{attribute 'GeneratedUsingTerminal: KL2819'}
{attribute addProperty BoxType "KL2819"}
{attribute addProperty Id "Channel_1AT %Q*Channel_2EC3E8CA0"}
{attribute addProperty CRC "685127745"}
{attribute addProperty Size "0"}
TYPE KL2819_28D63841 :
STRUCT
	{attribute addProperty Name "Channel_1"}
	Channel_1 : Channel_2EC3E8CA;
END_STRUCT
END_TYPE

(* stored: Version 1.2.0.0, ProductVersion 3.1.4024.9
   DUT KL2819_28D63841: Id {c018a0b4-27ec-4fd0-a0d6-2034c829f223} *)
